Yaskawa INFORM job: TWIN_SKRZYNIA_5340_0_STOPNI_1OBR.JBI

/JOB
//NAME TWIN_SKRZYNIA_5340_0_STOPNI_1OBR
///FOLDERNAME 02-SKRZYNIE_JOBS
//POS
///NPOS 402,402,0,35,0,0
///TOOL 0
///POSTYPE PULSE
///PULSE
C00000=1055,-24125,84372,288,19725,204
C00001=1055,-24125,84372,288,19725,204
C00002=0,-15438,65714,0,-68532,0
C00003=25524,-25821,36823,19654,-58495,38520
C00004=23988,-24960,37134,18595,-57837,38812
C00005=22822,-23954,37534,17811,-57199,39017
C00006=22935,-24057,37491,17887,-57262,38997
C00007=20006,-24258,37408,15644,-56932,39751
C00008=24402,-25289,37013,18874,-58060,38740
C00009=22585,-24665,40358,17164,-59622,30036
C00010=23477,-23257,40205,18030,-58646,29630
C00011=22519,-22398,40568,17384,-58125,29795
C00012=22700,-22567,40495,17506,-58225,29764
C00013=19339,-22794,40398,14955,-57865,30607
C00014=24825,-24328,39798,18931,-59350,29401
C00015=32755,-32613,25711,29640,-48730,33694
C00016=25632,-30899,26166,23992,-46203,35378
C00017=24264,-29862,26497,22996,-45413,35639
C00018=24403,-29974,26459,23097,-45496,35612
C00019=20575,-30233,26374,19602,-44891,36810
C00020=26556,-31526,25988,24663,-46720,35206
C00021=30846,-32795,25752,28021,-48338,30427
C00022=24953,-30697,26306,23444,-45946,31743
C00023=23937,-29910,26558,22702,-45353,31936
C00024=24039,-29993,26530,22778,-45414,31916
C00025=20322,-30240,26449,19379,-44834,33080
C00026=25997,-31433,26093,24205,-46535,31545
C00027=26028,-43665,26580,-39946,8682,24640
C00028=27956,-30595,53065,-101898,6609,54413
C00029=26028,-43663,26580,-39944,8677,24639
C00030=38784,-34544,25404,33956,-51320,34445
C00031=29266,-32676,25756,26732,-47889,36488
C00032=25734,-31262,26119,24020,-46377,37252
C00033=24289,-30200,26441,22967,-45549,37525
C00034=24367,-30262,26420,23025,-45594,37511
C00035=20043,-30544,26331,19080,-44922,38860
C00036=26573,-31816,25967,24631,-46839,37095
C00037=27817,-32566,25782,25532,-47502,36865
C00038=25779,-31294,26110,24054,-46400,37243
C00039=24344,-30243,26427,23007,-45578,37515
C00040=24432,-30312,26405,23072,-45630,37498
C00041=20021,-30599,26315,19050,-44944,38872
C00042=26262,-31616,26021,24405,-46667,37153
C00043=27439,-32346,25835,25259,-47302,36935
C00044=25570,-31108,26163,23910,-46262,37277
C00045=24581,-30384,26384,23190,-45695,37464
C00046=24689,-30466,26358,23269,-45758,37444
C00047=20001,-30771,26264,18999,-45026,38899
C00048=26308,-31607,26026,24448,-46671,37139
C00049=27526,-32360,25834,25329,-47326,36914
C00050=24269,-40076,6479,29767,-34177,34232
C00051=22958,-37632,10123,27061,-35370,35326
C00052=22703,-41294,1722,31272,-29953,33282
C00053=19440,-41515,1663,27208,-29122,34832
C00054=25465,-43501,1200,33269,-31905,32752
C00055=87177,-39066,-1236,81808,-72661,19198
C00056=4794,-34097,38974,4189,-31824,-1302
C00057=4794,-34097,38974,4189,13412,-1302
C00058=11237,-37131,38982,-12694,5333,8253
C00059=6591,-33902,35532,5956,-1761,-1932
C00060=10065,-33530,28876,9373,-31104,-3154
C00061=31877,-32319,25770,29025,-48287,33360
C00062=24706,-30765,26196,23236,-45867,35119
C00063=23652,-29939,26460,22464,-45250,35320
C00064=23742,-30013,26436,22530,-45305,35302
C00065=19630,-30281,26348,18756,-44677,36597
C00066=26056,-31710,25928,24219,-46631,34863
C00067=38095,-40136,7813,41252,-44156,24924
C00068=33231,-38681,8176,37792,-41757,25918
C00069=31538,-37640,8473,36716,-40716,26179
C00070=31687,-37737,8444,36811,-40809,26155
C00071=27389,-38154,8322,32773,-39589,27627
C00072=33834,-39023,8084,38175,-42120,25821
C00073=4801,-35772,25187,4594,-28023,-1125
C00074=-1002,-39861,25115,1795,-37402,-69601
C00075=-1001,-39858,25114,1795,-37402,0
C00076=6591,-33902,35532,5956,-1761,-1932
C00077=6592,-33900,35531,103508,-35512,-26314
C00078=-99253,-13690,44082,59847,13407,-31313
C00079=-85045,-36869,-4353,28502,-22832,-52282
C00080=-92346,-18713,13565,21110,-22545,-55257
C00081=-85370,-14218,16934,32905,-23649,-60330
C00082=-84150,-13282,17685,34842,-23935,-61163
C00083=-82877,-12536,18624,36445,-24482,-61818
C00084=-83784,-13116,17825,35378,-24051,-61391
C00085=-85049,-11554,19196,33922,-23396,-60809
C00086=-84150,-13282,17685,34842,-23935,-61163
C00087=-85732,-21202,11427,30682,-24763,-59235
C00088=-84559,-15616,15722,33768,-24118,-60665
C00089=-84150,-13282,17685,34842,-23935,-61163
C00090=-83260,-12880,18034,36130,-24218,-61709
C00091=-84150,-13282,17685,34842,-23935,-61163
C00092=-85365,-11775,19006,33430,-23307,-60600
C00093=-84150,-13282,17685,34842,-23935,-61163
C00094=-85786,-16909,14677,31743,-23900,-59790
C00095=-84150,-13282,17685,34842,-23935,-61163
C00096=-83215,-12861,18051,36194,-24233,-61735
C00097=-84150,-13282,17685,34842,-23935,-61163
C00098=-85327,-11825,18959,33476,-23327,-60618
C00099=-84150,-13282,17685,34842,-23935,-61163
C00100=-87841,-18519,13420,28367,-23534,-58339
C00101=-84150,-13282,17685,34842,-23935,-61163
C00102=-83292,-12894,18020,36083,-24208,-61688
C00103=-84150,-13282,17685,34842,-23935,-61163
C00104=-85185,-12008,18799,33646,-23400,-60687
C00105=-84150,-13282,17685,34842,-23935,-61163
C00106=-86371,-18277,13606,30568,-23951,-59265
C00107=-84345,-13370,17612,34554,-23873,-61041
C00108=-83240,-12871,18042,36158,-24225,-61720
C00109=-84345,-13370,17612,34554,-23873,-61041
C00110=-85365,-12110,18711,33368,-23345,-60568
C00111=-84345,-13370,17612,34554,-23873,-61041
C00112=-86191,-19647,12567,30467,-24278,-59187
C00113=-84345,-13372,17610,34552,-23873,-61039
C00114=-83096,-12807,18098,36363,-24268,-61804
C00115=-84345,-13372,17610,34552,-23873,-61039
C00116=-85268,-12232,18600,33480,-23393,-60612
C00117=-84345,-13372,17610,34552,-23873,-61039
C00118=-84814,-16043,15376,33312,-24093,-60464
C00119=-84104,-13265,17702,34906,-23948,-61189
C00120=-82960,-12743,18153,36555,-24313,-61887
C00121=-84104,-13265,17702,34906,-23948,-61189
C00122=-84979,-12194,18635,33901,-23496,-60788
C00123=-84104,-13265,17702,34906,-23948,-61189
C00124=-86610,-16845,14732,30573,-23614,-59301
C00125=-84104,-13265,17702,34906,-23948,-61189
C00126=-82793,-12667,18222,36790,-24370,-61986
C00127=-84104,-13265,17702,34906,-23948,-61189
C00128=-84888,-12305,18537,34004,-23540,-60830
C00129=-84104,-13265,17702,34906,-23948,-61189
C00130=-83806,-19585,12613,33764,-25080,-60559
C00131=-83675,-13072,17868,35530,-24083,-61453
C00132=-82553,-12556,18319,37130,-24451,-62127
C00133=-83675,-13072,17868,35530,-24083,-61453
C00134=-84378,-12223,18610,34735,-23716,-61138
C00135=-83675,-13072,17868,35530,-24083,-61453
C00136=-87149,-17993,13826,29513,-23647,-58830
C00137=-84104,-13265,17702,34906,-23948,-61189
C00138=-82640,-12594,18285,37014,-24425,-62079
C00139=-84104,-13265,17702,34906,-23948,-61189
C00140=-84792,-12429,18430,34119,-23592,-60877
C00141=-84104,-13265,17702,34906,-23948,-61189
C00142=-83583,-9185,30892,23668,-36042,-57025
C00143=-85789,-8328,35795,20592,-37093,-55378
C00144=-85786,-16735,14816,31782,-23869,-59812
C00145=-84103,-13263,17702,34906,-23947,-61191
C00146=-83225,-12865,18046,36177,-24227,-61729
C00147=-84103,-13263,17702,34906,-23947,-61191
C00148=-84774,-12447,18412,34138,-23599,-60886
C00149=-84103,-13263,17702,34906,-23947,-61191
C00150=-86149,-16246,6730,18897,-35239,-57128
C00151=-86244,-15289,7532,18875,-35060,-57127
C00152=-85361,-14893,7870,19824,-35193,-57574
C00153=-86244,-15289,7532,18875,-35060,-57127
C00154=-86889,-14409,8282,18264,-34784,-56850
C00155=-86244,-15289,7532,18875,-35060,-57127
C00156=-90262,-21765,2389,14114,-35574,-54847
C00157=-90262,-21765,2389,28730,-17672,-54847
C00158=-89967,-19086,25635,28730,-17672,-54847
C00159=568,-24029,84339,168,19981,112
C00160=568,-24677,83015,164,20405,113
C00161=101153,-24598,83176,165,20353,113
C00162=101153,-24598,83176,165,20353,113
C00163=89967,-19086,25635,-28730,-17672,54847
C00164=90262,-21765,2389,-28730,-17672,54847
C00165=86932,-18662,4771,-17876,-35519,56628
C00166=86578,-15436,7408,-18515,-35011,56957
C00167=85428,-14922,7844,-19753,-35183,57541
C00168=84405,-14447,8250,-20842,-35348,58054
C00169=85428,-14922,7844,-19753,-35183,57541
C00170=86134,-13973,8661,-19091,-34881,57237
C00171=85428,-14922,7844,-19753,-35183,57541
C00172=85786,-16735,14816,-31782,-23869,59812
C00173=83514,-12996,17929,-35760,-24132,61552
C00174=82296,-12429,18424,-37488,-24534,62281
C00175=83514,-12996,17929,-35760,-24132,61552
C00176=84266,-12085,18725,-34910,-23738,61214
C00177=83514,-12996,17929,-35760,-24132,61552
C00178=87323,-6914,39851,-18853,-38149,44508
C00179=83118,-12818,18089,-36330,-24263,61791
C00180=81969,-12276,18566,-37944,-24648,62472
C00181=83118,-12818,18089,-36330,-24263,61791
C00182=83927,-11846,18941,-35423,-23842,61433
C00183=83118,-12818,18089,-36330,-24263,61791
C00184=83806,-19585,12613,-33764,-25080,60559
C00185=83148,-12832,18077,-36287,-24254,61773
C00186=81889,-12236,18598,-38058,-24676,62520
C00187=83148,-12832,18077,-36287,-24254,61773
C00188=83900,-11930,18867,-35446,-23862,61440
C00189=83148,-12832,18077,-36287,-24254,61773
C00190=86610,-16845,14732,-30573,-23614,59301
C00191=82493,-13239,17725,-37070,-24559,62089
C00192=81442,-12739,18159,-38529,-24915,62703
C00193=82493,-13239,17725,-37070,-24559,62089
C00194=83435,-12133,18689,-36040,-24063,61682
C00195=82493,-13239,17725,-37070,-24559,62089
C00196=84814,-16043,15376,-33312,-24093,60464
C00197=82555,-13613,17404,-36910,-24580,62015
C00198=81369,-13053,17885,-38558,-24979,62709
C00199=82555,-13613,17404,-36910,-24580,62015
C00200=83568,-12431,18429,-35805,-24046,61580
C00201=82555,-13613,17404,-36910,-24580,62015
C00202=86191,-19647,12567,-30467,-24278,59187
C00203=82500,-13648,17375,-36975,-24607,62039
C00204=81594,-13224,17740,-38236,-24911,62571
C00205=82500,-13648,17375,-36975,-24607,62039
C00206=83449,-12543,18332,-35941,-24104,61633
C00207=82500,-13648,17375,-36975,-24607,62039
C00208=86371,-18277,13606,-30568,-23951,59265
C00209=82904,-13790,17251,-36416,-24470,61808
C00210=81796,-13275,17692,-37971,-24838,62464
C00211=82904,-13790,17251,-36416,-24470,61808
C00212=83696,-12867,18046,-35547,-24051,61466
C00213=82904,-13790,17251,-36416,-24470,61808
C00214=87841,-18519,13420,-28367,-23534,58339
C00215=82748,-13879,17174,-36603,-24542,61883
C00216=81789,-13434,17554,-37946,-24861,62449
C00217=82748,-13879,17174,-36603,-24542,61883
C00218=83603,-12888,18026,-35668,-24086,61514
C00219=82748,-13879,17174,-36603,-24542,61883
C00220=85786,-16909,14677,-31743,-23900,59790
C00221=82339,-14116,16972,-37087,-24733,62079
C00222=81557,-13752,17280,-38171,-24994,62536
C00223=82339,-14116,16972,-37087,-24733,62079
C00224=83390,-12909,18006,-35951,-24172,61633
C00225=82339,-14116,16972,-37087,-24733,62079
C00226=85732,-21202,11427,-30682,-24763,59235
C00227=82398,-14365,16763,-36952,-24745,62014
C00228=81340,-13876,17176,-38416,-25096,62632
C00229=82398,-14365,16763,-36952,-24745,62014
C00230=83629,-12951,17972,-35620,-24090,61491
C00231=82398,-14365,16763,-36952,-24745,62014
C00232=92346,-18713,13565,-21110,-22545,55257
C00233=82794,-13980,17083,-36511,-24538,61844
C00234=81697,-13472,17516,-38043,-24902,62488
C00235=82794,-13980,17083,-36511,-24538,61844
C00236=83767,-12847,18056,-35444,-24023,61424
C00237=82794,-13980,17083,-36511,-24538,61844
C00238=85045,-36869,-4353,-28502,-22832,52282
C00239=69856,-53931,-13446,-33557,-28911,29591
C00240=73943,-28815,39553,-16801,-45089,19004
C00241=73943,-28815,39553,-16801,-45089,19004
C00242=0,-24029,84339,0,19981,0
C00243=0,-24029,84339,0,19981,0
C00244=0,-52280,40443,0,6876,0
C00245=63961,-36661,14391,66570,-58199,13439
C00246=50233,-31965,16595,55443,-54435,15843
C00247=47147,-32819,12541,55607,-51124,17230
C00248=46896,-37872,871,62973,-46008,11193
C00249=54160,-39955,137,66075,-50361,10746
C00250=0,-52280,40443,0,6876,0
C00251=0,-52280,40443,1,6876,0
C00252=42978,-45587,7631,48214,-41849,18034
C00253=34615,-32719,24207,35617,-45539,22507
C00254=46734,-24688,30880,50025,-55713,21863
C00255=45059,-39151,-3508,69830,-41334,11649
C00256=32474,-45233,-13338,65386,-28486,22104
C00257=59828,-44646,-5405,72855,-48572,12139
C00258=0,-38761,66314,0,-763,0
C00259=0,-44757,54667,0,2744,0
C00260=40382,-38226,12225,48505,-40693,16039
C00261=55481,-27484,23768,62968,-54833,11978
C00262=49796,-26552,24209,59898,-51910,12564
C00263=49435,-31346,12259,54968,-55893,13137
C00264=55330,-33748,11238,57660,-59334,12681
C00265=78664,-24436,10378,82837,-79111,12029
C00266=75189,-23065,11287,81851,-76948,11927
C00267=75189,-45249,11287,81851,-38847,11927
C00268=29880,-45249,11287,43145,-11324,11927
C00269=0,-24029,84339,0,19981,0
C00270=0,-24026,84338,1,19977,2
C00271=4264,-34194,25387,4006,-26954,-29436
C00272=1,-24024,84337,2,19973,1
C00273=1,-24024,84337,2,19973,1
C00274=3796,-57671,22373,2336,-25309,-753
C00275=52632,-34554,16626,51161,-63050,5622
C00276=59461,-32779,9832,66317,-58406,17312
C00277=52698,-27865,19111,60288,-56542,14852
C00278=51544,-17445,41630,51689,-64712,19351
C00279=62932,-33588,12189,66848,-61063,18031
C00280=1,-24024,84337,2,19973,1
C00281=1,-24024,84337,2,19973,1
C00282=57188,-41777,19973,48132,-58706,4905
C00283=55566,-48748,-16991,79805,-45048,-6941
C00284=49908,-48716,-25784,90749,-41340,-3650
C00285=44252,-47412,-25530,90709,-37744,-4391
C00286=43421,-46995,-25379,90839,-37219,-4572
C00287=55479,-50244,-26473,91085,-44870,-3042
C00288=12119,-24859,71505,13236,4440,2633
C00289=-91085,-34291,10385,1908,-24348,-42097
C00290=-86191,-19647,12567,30467,-24278,-59187
C00291=-99148,-11667,19101,-13975,-20192,-40187
C00292=-98206,-11518,19604,-10142,-20308,-41629
C00293=-99474,-20389,12397,-11593,-22150,-41069
C00294=0,-52280,40443,0,6876,0
C00295=85348,-24204,23536,-13963,-15515,44275
C00296=84670,-17015,14597,-33277,-24304,60423
C00297=96971,-12584,18294,8365,-19955,42614
C00298=97182,-12918,18001,8747,-20027,42449
C00299=96230,-24528,9149,6144,-22576,43630
C00300=0,-52280,40443,0,6876,0
C00301=0,-52280,40443,0,6876,0
C00302=-90140,-60305,18108,-2708,1721,-7625
C00303=-95594,-27428,6866,-4663,-19832,-42154
C00304=-99356,-13410,18355,-15385,-17730,-37479
C00305=-99405,-10878,20508,-15853,-17333,-37255
C00306=-99132,-10804,20575,-15274,-17279,-37502
C00307=-99132,-3482,39129,-10940,-24351,-39674
C00308=-98851,-3328,38974,-10588,-24101,-39807
C00309=-100183,-18601,14070,-16273,-18800,-37146
C00310=-90140,-60305,18108,-2708,1721,-7625
C00311=0,-52280,40443,0,6876,0
C00312=84259,-57935,27522,-3761,3673,6310
C00313=86507,-39672,4297,-27618,-16640,46340
C00314=70477,-27878,7073,-45786,-32339,64941
C00315=84043,-16293,15174,-34312,-24409,60872
C00316=94507,-13191,17794,-563,-19874,46473
C00317=99154,-17369,4403,32227,-9753,28926
C00318=99154,-17369,4403,32227,-9753,28926
C00319=98946,-17182,4556,31649,-9649,29182
C00320=100388,-17987,13832,15751,-21517,39479
C00321=86507,-39672,4297,-27618,-16640,46340
C00322=84259,-57935,27522,-3761,3673,6310
C00323=0,-52280,40443,0,6876,0
C00324=0,-27933,77061,0,20812,0
C00325=0,-27933,77061,0,20812,0
C00326=0,-52280,40443,0,6876,0
C00327=-91970,-60791,14435,-3343,512,-9412
C00328=-99196,-15868,16098,-13748,-19297,-38710
C00329=-99196,-15868,16098,-13748,-19297,-38710
C00330=-99196,-15868,16098,-13748,-19297,-38710
C00331=-85815,-11758,19597,31748,-21097,-58265
C00332=-87383,-11883,19487,26986,-20206,-56250
C00333=-99562,-16264,15781,-14410,-19427,-38431
C00334=-99196,-15868,16098,-13748,-19297,-38710
C00335=-91970,-60791,14435,-3343,512,-9412
C00336=0,-52280,40443,0,6876,0
C00337=91083,-60784,14823,-9043,-825,15173
C00338=83869,-19403,12921,-33769,-24740,60260
C00339=83869,-19403,12921,-33769,-24740,60260
C00340=83420,-14897,16486,-35538,-24144,61113
C00341=90535,-11845,19652,-14037,-20800,51549
C00342=90317,-11662,19878,-14346,-20882,51648
C00343=95871,-14889,15992,4901,-19605,43825
C00344=83869,-19403,12921,-33769,-24740,60260
C00345=91083,-60784,14823,-9043,-825,15173
C00346=0,-52280,40443,0,6876,0
C00347=-91526,-60598,16699,7584,176,-13289
C00348=-94392,-6553,48683,5805,-47321,-49764
C00349=-88951,-345,54953,10686,-47392,-51569
C00350=-88172,5833,62122,11322,-47753,-51785
C00351=-90949,-14015,9500,8834,-34399,-51934
C00352=-84917,-15593,15742,33275,-23984,-60461
C00353=-81669,-15982,15425,37506,-25258,-62202
C00354=-79867,-25377,9541,37586,-25936,-59971
C00355=-91415,-60262,16631,7870,-73,-13734
C00356=24,-24029,84339,7,19981,5
C00357=160,-24029,84339,47,19981,32
C00358=99096,-24029,84339,47,19981,32
C00359=99096,-24029,84339,47,19981,32
C00360=89967,-19086,25635,-28730,-17672,54847
C00361=85786,-16735,14816,-31782,-23869,59812
C00362=83492,-14473,16674,-35480,-24338,61406
C00363=82709,-11470,19305,-37370,-24374,62232
C00364=85293,-13629,8874,-19696,-34851,57583
C00365=85505,-16299,6686,-19564,-35388,57437
C00366=89967,-19086,25635,-28730,-17672,54847
C00367=568,-24029,84339,168,19981,112
C00368=568,-24029,84339,168,19981,112
C00369=-91970,-60791,14435,-3343,512,-9412
C00370=-86948,-23217,10819,28314,-23349,-56438
C00371=-85895,-16522,15767,31843,-22281,-58087
C00372=-93643,1708,52973,2937,-38210,-34777
C00373=-93409,-737,47229,3345,-36106,-34967
C00374=-86145,-24679,9854,29028,-23971,-56682
C00375=-100471,-58311,4157,14142,-4822,-27614
C00376=-68517,-58311,4157,14142,-4822,-27614
C00377=0,-52280,40443,0,6876,0
C00378=91083,-60784,14823,-9043,-825,15173
C00379=83869,-19403,12921,-33769,-24740,60260
C00380=82620,-18743,14708,-32942,-26226,58979
C00381=83315,-11405,20766,-33572,-24860,59408
C00382=83326,-11144,20997,-33599,-24827,59423
C00383=84798,-22668,11879,-29033,-26372,57255
C00384=91083,-60784,14823,-9043,-825,15173
C00385=0,-52280,40443,0,6876,0
C00386=-6369,-39206,65423,-4801,-482,2563
C00387=-97287,-29142,12714,-8673,-22288,-37832
C00388=-86191,-19647,12567,30467,-24278,-59187
C00389=-85671,-16302,15857,30808,-24404,-58999
C00390=-99965,-10410,22406,-14600,-22538,-38834
C00391=-95758,-10871,21797,-1120,-21702,-44724
C00392=-87910,-17792,15835,25414,-24996,-56048
C00393=-97287,-29142,12714,-8673,-22288,-37832
C00394=0,-52280,40443,0,6876,0
C00395=92301,-25634,22749,2368,-15645,37646
C00396=83738,-18329,13570,-34202,-24868,60772
C00397=90096,-13099,18146,-15422,-20883,52700
C00398=93330,-13245,17928,-4627,-20146,48105
C00399=80226,-20465,12178,-39626,-27411,62762
C00400=92301,-25634,22749,2368,-15645,37646
C00401=0,-52280,40443,0,6876,0
BC00000=413138
BC00001=413138
BC00002=413138
BC00003=413134
BC00004=413134
BC00005=413134
BC00006=413134
BC00007=413134
BC00008=413134
BC00009=474623
BC00010=474628
BC00011=474628
BC00012=474628
BC00013=474628
BC00014=474628
BC00015=522849
BC00016=522849
BC00017=522849
BC00018=522849
BC00019=522849
BC00020=522849
BC00021=586045
BC00022=586045
BC00023=586045
BC00024=586045
BC00025=586045
BC00026=586045
BC00027=479622
BC00028=618860
BC00029=673957
BC00030=663090
BC00031=663090
BC00032=663090
BC00033=663090
BC00034=663090
BC00035=663090
BC00036=663090
BC00037=708270
BC00038=708270
BC00039=708270
BC00040=708270
BC00041=708270
BC00042=708270
BC00043=770184
BC00044=770184
BC00045=770184
BC00046=770184
BC00047=770184
BC00048=770184
BC00049=823730
BC00050=829967
BC00051=829969
BC00052=829970
BC00053=829970
BC00054=829970
BC00055=838761
BC00056=740349
BC00057=687700
BC00058=771943
BC00059=861898
BC00060=900223
BC00061=904141
BC00062=901229
BC00063=901229
BC00064=901229
BC00065=901229
BC00066=901229
BC00067=949836
BC00068=949836
BC00069=949836
BC00070=949836
BC00071=949836
BC00072=965197
BC00073=941874
BC00074=915598
BC00075=930961
BC00076=861898
BC00077=861901
BC00078=861901
BC00079=931504
BC00080=963634
BC00081=963631
BC00082=963631
BC00083=963631
BC00084=963631
BC00085=963631
BC00086=963631
BC00087=902188
BC00088=902188
BC00089=902188
BC00090=902188
BC00091=902188
BC00092=902188
BC00093=902188
BC00094=840744
BC00095=840744
BC00096=840744
BC00097=840744
BC00098=840744
BC00099=840744
BC00100=779300
BC00101=779300
BC00102=779300
BC00103=779300
BC00104=779300
BC00105=779300
BC00106=717855
BC00107=717855
BC00108=717855
BC00109=717855
BC00110=717855
BC00111=717855
BC00112=656405
BC00113=656405
BC00114=656405
BC00115=656405
BC00116=656405
BC00117=656405
BC00118=594961
BC00119=594961
BC00120=594961
BC00121=594961
BC00122=594961
BC00123=594961
BC00124=533517
BC00125=533517
BC00126=533517
BC00127=533517
BC00128=533517
BC00129=533517
BC00130=472073
BC00131=472073
BC00132=472073
BC00133=472073
BC00134=472073
BC00135=472073
BC00136=410629
BC00137=410629
BC00138=410629
BC00139=410629
BC00140=410629
BC00141=410629
BC00142=410629
BC00143=349186
BC00144=349186
BC00145=349186
BC00146=349186
BC00147=349186
BC00148=349186
BC00149=349186
BC00150=336469
BC00151=336469
BC00152=336469
BC00153=336469
BC00154=336469
BC00155=336469
BC00156=336469
BC00157=336469
BC00158=336469
BC00159=336469
BC00160=511557
BC00161=512005
BC00162=363797
BC00163=336469
BC00164=336469
BC00165=337415
BC00166=337415
BC00167=337415
BC00168=337415
BC00169=337415
BC00170=337415
BC00171=337415
BC00172=349186
BC00173=350137
BC00174=350137
BC00175=350137
BC00176=350137
BC00177=350137
BC00178=410629
BC00179=411580
BC00180=411580
BC00181=411580
BC00182=411580
BC00183=411580
BC00184=472073
BC00185=473025
BC00186=473025
BC00187=473025
BC00188=473025
BC00189=473025
BC00190=533517
BC00191=534468
BC00192=534468
BC00193=534468
BC00194=534468
BC00195=534468
BC00196=594961
BC00197=594961
BC00198=594961
BC00199=594961
BC00200=594961
BC00201=594961
BC00202=656405
BC00203=657350
BC00204=657350
BC00205=657350
BC00206=657350
BC00207=657350
BC00208=717855
BC00209=718799
BC00210=718799
BC00211=718799
BC00212=718799
BC00213=718799
BC00214=779300
BC00215=780245
BC00216=780245
BC00217=780245
BC00218=780245
BC00219=780245
BC00220=840744
BC00221=841691
BC00222=841691
BC00223=841691
BC00224=841691
BC00225=841691
BC00226=902188
BC00227=903136
BC00228=903136
BC00229=903136
BC00230=903136
BC00231=903136
BC00232=963634
BC00233=963633
BC00234=963633
BC00235=963633
BC00236=963633
BC00237=963633
BC00238=931504
BC00239=861901
BC00240=861901
BC00241=881624
BC00242=769966
BC00243=769966
BC00244=716865
BC00245=668657
BC00246=668657
BC00247=668657
BC00248=717171
BC00249=717171
BC00250=716865
BC00251=800897
BC00252=908887
BC00253=899019
BC00254=895607
BC00255=945882
BC00256=955598
BC00257=945882
BC00258=840120
BC00259=538973
BC00260=485226
BC00261=456696
BC00262=456696
BC00263=417276
BC00264=417276
BC00265=493986
BC00266=514306
BC00267=514306
BC00268=514306
BC00269=493986
BC00270=797003
BC00271=895791
BC00272=812362
BC00273=476651
BC00274=522561
BC00275=566531
BC00276=593948
BC00277=593948
BC00278=529848
BC00279=529848
BC00280=461290
BC00281=663315
BC00282=778314
BC00283=778312
BC00284=778312
BC00285=778312
BC00286=838222
BC00287=838222
BC00288=566410
BC00289=679663
BC00290=656405
BC00291=656405
BC00292=717855
BC00293=717855
BC00294=717855
BC00295=662303
BC00296=657350
BC00297=657350
BC00298=718803
BC00299=718803
BC00300=717855
BC00301=792672
BC00302=792672
BC00303=896850
BC00304=895720
BC00305=895720
BC00306=957178
BC00307=957178
BC00308=978461
BC00309=957178
BC00310=792672
BC00311=792672
BC00312=792672
BC00313=887446
BC00314=903126
BC00315=903126
BC00316=903126
BC00317=964577
BC00318=976097
BC00319=993812
BC00320=964577
BC00321=887446
BC00322=792672
BC00323=792672
BC00324=700249
BC00325=546214
BC00326=546214
BC00327=546211
BC00328=546211
BC00329=406776
BC00330=406776
BC00331=406778
BC00332=468200
BC00333=468200
BC00334=546211
BC00335=546211
BC00336=546214
BC00337=546214
BC00338=507604
BC00339=410782
BC00340=410782
BC00341=410782
BC00342=472720
BC00343=472720
BC00344=507604
BC00345=546214
BC00346=546214
BC00347=516757
BC00348=383716
BC00349=349186
BC00350=349186
BC00351=336469
BC00352=349186
BC00353=410629
BC00354=416512
BC00355=515801
BC00356=520018
BC00357=474013
BC00358=474013
BC00359=403108
BC00360=336469
BC00361=349186
BC00362=349186
BC00363=349186
BC00364=337415
BC00365=337415
BC00366=336469
BC00367=336469
BC00368=428401
BC00369=546211
BC00370=591088
BC00371=591088
BC00372=591088
BC00373=531116
BC00374=529640
BC00375=529640
BC00376=529640
BC00377=529640
BC00378=546214
BC00379=589919
BC00380=595627
BC00381=595627
BC00382=534177
BC00383=534177
BC00384=546214
BC00385=529640
BC00386=651195
BC00387=765890
BC00388=777968
BC00389=778453
BC00390=779252
BC00391=840748
BC00392=840748
BC00393=765890
BC00394=717855
BC00395=741100
BC00396=780224
BC00397=780222
BC00398=841743
BC00399=841743
BC00400=741100
BC00401=717855
///POSTYPE BASE
///RECTAN
///RCONF 0,0,0,0,0,0,0,0,0,0,0,0,0,0,0,0,0,0,0,0,0,0,0,0
P00006=-2.449,0.031,8.825,0.0000,0.0000,0.0000
///RCONF 1,0,0,0,0,0,0,0,0,0,0,0,0,0,0,0,0,0,0,0,0,0,0,0
P00100=-0.081,2.558,4.482,0.0000,0.0000,0.0000
P00101=0.030,-2.286,2.993,0.0000,0.0000,0.0000
P00102=-0.005,-1.108,1.644,0.0000,0.0000,0.0000
P00103=-0.094,-3.400,4.200,0.0000,0.0000,0.0000
P00104=0.043,-2.127,5.826,0.0000,0.0000,0.0000
P00105=-0.043,0.662,5.286,0.0000,0.0000,0.0000
P00106=-0.018,-2.519,0.237,0.0000,0.0000,0.0000
P00107=-0.008,-4.537,-4.500,0.0000,0.0000,0.0000
P00108=0.014,-3.040,2.637,0.0000,0.0000,0.0000
P00109=0.017,-3.622,2.341,0.0000,0.0000,0.0000
P00300=-0.036,-1.505,2.318,0.0000,0.0000,0.0000
///RCONF 0,0,0,0,0,0,0,0,0,0,0,0,0,0,0,0,0,0,0,0,0,0,0,0
P00301=0.005,-4.708,-4.628,0.0000,0.0000,0.0000
P00302=0.052,-2.937,-4.426,0.0000,0.0000,0.0000
P00303=-0.004,-1.437,-4.584,0.0000,0.0000,0.0000
P00304=0.028,-1.666,-4.234,0.0000,0.0000,0.0000
P00305=-0.003,-1.920,-3.501,0.0000,0.0000,0.0000
P00306=0.015,-2.252,-3.054,0.0000,0.0000,0.0000
P00307=0.019,-2.151,-5.077,0.0000,0.0000,0.0000
P00308=-0.003,-2.092,-4.888,0.0000,0.0000,0.0000
P00309=-0.040,-2.205,-4.992,0.0000,0.0000,0.0000
P00310=-0.006,-2.490,-5.925,0.0000,0.0000,0.0000
P00311=-0.007,-2.079,-5.307,0.0000,0.0000,0.0000
P00350=11.519,-0.008,1.149,0.0000,0.0000,0.0000
P00351=13.563,-0.027,-0.653,0.0000,0.0000,0.0000
P00352=13.252,-0.027,-0.827,0.0000,0.0000,0.0000
P00353=10.971,-0.082,0.776,0.0000,0.0000,0.0000
P00354=-0.024,2.508,-1.824,0.0000,0.0000,0.0000
P00355=-0.001,2.528,-1.131,0.0000,0.0000,0.0000
P00356=-0.034,2.921,-0.262,0.0000,0.0000,0.0000
P00357=0.003,3.386,-0.091,0.0000,0.0000,0.0000
P00358=0.014,3.037,-0.020,0.0000,0.0000,0.0000
P00359=-0.005,2.731,0.912,0.0000,0.0000,0.0000
P00360=-0.011,3.412,0.438,0.0000,0.0000,0.0000
P00361=0.018,3.050,1.253,0.0000,0.0000,0.0000
//INST
///DATE 2024/12/12 11:36
///ATTR SC,RW
///GROUP1 RB1,BS1
NOP
CALL JOB:MOVE_INTO_TUNNEL
MOVJ C00000 BC00000 VJ=30.00
'------------------------
'------------------------
'SPOINA SRODEK DOL
'------------------------
'------------------------
'POMIAR DO WYJ!! PRZEROBIC NA STD
MOVJ C00001 BC00001 VJ=40.00
MOVJ C00002 BC00002 VJ=40.00
'W3P
MOVJ C00003 BC00003 VJ=20.00 PL=0
MOVL C00004 BC00004 V=166.7 PL=0
REFP 3 C00005 BC00005
CALL JOB:SEARCH-R1
SET P0100 P0006
SFTON P0100
MOVL C00006 BC00006 V=66.7 PL=0
REFP 3 C00007 BC00007
CALL JOB:SEARCH-R1
SET P0100 P0006
SFTON P0100
MOVL C00008 BC00008 V=333.3 PL=0
SFTOF
'W3L
MOVL C00009 BC00009 V=666.7
MOVL C00010 BC00010 V=166.7 PL=0
REFP 3 C00011 BC00011
CALL JOB:SEARCH-R1
SET P0101 P0006
SFTON P0101
MOVL C00012 BC00012 V=166.7 PL=0
REFP 3 C00013 BC00013
CALL JOB:SEARCH-R1
SET P0101 P0006
SFTON P0101
MOVL C00014 BC00014 V=333.3 PL=0
SFTOF
'W9P
MOVL C00015 BC00015 V=666.7
MOVL C00016 BC00016 V=166.7
REFP 3 C00017 BC00017
CALL JOB:SEARCH-R1
SET P0102 P0006
SFTON P0102
MOVL C00018 BC00018 V=166.7 PL=0
REFP 3 C00019 BC00019
CALL JOB:SEARCH-R1
SET P0102 P0006
SFTON P0102
MOVL C00020 BC00020 V=333.3 PL=0
'W9L
MOVL C00021 BC00021 V=666.7
MOVL C00022 BC00022 V=166.7
REFP 3 C00023 BC00023
CALL JOB:SEARCH-R1
SET P0103 P0006
SFTON P0103
MOVL C00024 BC00024 V=166.7 PL=0
REFP 3 C00025 BC00025
CALL JOB:SEARCH-R1
SET P0103 P0006
SFTON P0103
MOVL C00026 BC00026 V=333.3 PL=0
'PRZEJAZ NAD BELKA
MOVL C00027 BC00027 V=666.7
MOVJ C00028 BC00028 VJ=40.00
MOVJ C00029 BC00029 VJ=40.00
MOVJ C00030 BC00030 VJ=40.00
'W1P
MOVJ C00031 BC00031 VJ=20.00 PL=0
MOVL C00032 BC00032 V=166.7 PL=0
REFP 3 C00033 BC00033
CALL JOB:SEARCH-R1
SET P0104 P0006
SFTON P0104
MOVL C00034 BC00034 V=166.7 PL=0
REFP 3 C00035 BC00035
CALL JOB:SEARCH-R1
SET P0104 P0006
SFTON P0104
MOVL C00036 BC00036 V=333.3 PL=0
SFTOF
'W1L
MOVL C00037 BC00037 V=666.7
MOVL C00038 BC00038 V=166.7 PL=0
REFP 3 C00039 BC00039
CALL JOB:SEARCH-R1
SET P0105 P0006
SFTON P0105
MOVL C00040 BC00040 V=166.7 PL=0
REFP 3 C00041 BC00041
CALL JOB:SEARCH-R1
SET P0105 P0006
SFTON P0105
MOVL C00042 BC00042 V=333.3 PL=0
SFTOF
MOVL C00043 BC00043 V=666.7
'W10P
MOVL C00044 BC00044 V=166.7 PL=0
REFP 3 C00045 BC00045
CALL JOB:SEARCH-R1
SET P0106 P0006
SFTON P0106
MOVL C00046 BC00046 V=166.7 PL=0
REFP 3 C00047 BC00047
CALL JOB:SEARCH-R1
SET P0106 P0006
SFTON P0106
MOVL C00048 BC00048 V=333.3 PL=0
SFTOF
'W10L
MOVL C00049 BC00049 V=333.3
MOVL C00050 BC00050 V=166.7 PL=0
REFP 3 C00051 BC00051
CALL JOB:SEARCH-R1
SET P0107 P0006
SFTON P0107
MOVL C00052 BC00052 V=166.7 PL=0
REFP 3 C00053 BC00053
CALL JOB:SEARCH-R1
SET P0107 P0006
SFTON P0107
MOVL C00054 BC00054 V=333.3 PL=0
SFTOF
MOVL C00055 BC00055 V=333.3
'PRZEJAZD
MOVJ C00056 BC00056 VJ=50.00
MOVJ C00057 BC00057 VJ=50.00
MOVJ C00058 BC00058 VJ=60.00
MOVJ C00059 BC00059 VJ=60.00
MOVJ C00060 BC00060 VJ=60.00
MOVJ C00061 BC00061 VJ=60.00 PL=0
MOVL C00062 BC00062 V=166.7 PL=0
REFP 3 C00063 BC00063
CALL JOB:SEARCH-R1
SET P0108 P0006
SFTON P0108
MOVL C00064 BC00064 V=166.7 PL=0
REFP 3 C00065 BC00065
CALL JOB:SEARCH-R1
SET P0108 P0006
SFTON P0108
MOVL C00066 BC00066 V=333.3 PL=0
SFTOF
'W2P
'W2L
MOVL C00067 BC00067 V=666.7
MOVL C00068 BC00068 V=166.7 PL=0
REFP 3 C00069 BC00069
CALL JOB:SEARCH-R1
SET P0109 P0006
SFTON P0109
MOVL C00070 BC00070 V=166.7 PL=0
REFP 3 C00071 BC00071
CALL JOB:SEARCH-R1
SET P0109 P0006
SFTON P0109
MOVL C00072 BC00072 V=333.3 PL=0
MOVJ C00073 BC00073 VJ=20.00
SFTOF
CALL JOB:TWIN_5340_0ST_RAMA_PRZ_OBR1_POM
'.................
'.................
'.................
'PROG POMIARY RAMA PRZED
'.................
'.................
'.................
MOVJ C00074 BC00074 VJ=50.00
'------------------------
'------------------------
'PRAWA STRONA PROFIL GORA
'------------------------
'------------------------
MOVJ C00075 BC00075 VJ=50.00
MOVJ C00076 BC00076 VJ=50.00
MOVJ C00077 BC00077 VJ=50.00
MOVJ C00078 BC00078 VJ=20.00
MOVJ C00079 BC00079 VJ=50.00
'------------------------
'W14A L
'------------------------
SFTOF
MOVJ C00080 BC00080 VJ=50.00
MOVJ C00081 BC00081 VJ=30.00
MOVL C00082 BC00082 V=166.7 PL=0
REFP 3 C00083 BC00083
CALL JOB:SEARCH-R1
SET P0300 P0006
SFTON P0300
MOVL C00084 BC00084 V=166.7 PL=0
REFP 3 C00085 BC00085
CALL JOB:SEARCH-R1
SET P0300 P0006
SFTON P0300
MOVL C00086 BC00086 V=166.7 PL=0
SFTOF
'------------------------
'W14A P
'------------------------
SFTOF
MOVJ C00087 BC00087 VJ=50.00
MOVJ C00088 BC00088 VJ=50.00
MOVL C00089 BC00089 V=166.7 PL=0
REFP 3 C00090 BC00090
CALL JOB:SEARCH-R1
SET P0301 P0006
SFTON P0301
MOVL C00091 BC00091 V=166.7 PL=0
REFP 3 C00092 BC00092
CALL JOB:SEARCH-R1
SET P0301 P0006
SFTON P0301
MOVL C00093 BC00093 V=166.7 PL=0
SFTOF
'------------------------
'W19A L
'------------------------
SFTOF
MOVJ C00094 BC00094 VJ=50.00
MOVL C00095 BC00095 V=200.0 PL=0
REFP 3 C00096 BC00096
CALL JOB:SEARCH-R1
SET P0302 P0006
SFTON P0302
MOVL C00097 BC00097 V=166.7 PL=0
REFP 3 C00098 BC00098
CALL JOB:SEARCH-R1
SET P0302 P0006
SFTON P0302
MOVL C00099 BC00099 V=250.0 PL=0
SFTOF
'------------------------
'W19A P
'------------------------
SFTOF
MOVJ C00100 BC00100 VJ=50.00
MOVL C00101 BC00101 V=166.7 PL=0
REFP 3 C00102 BC00102
CALL JOB:SEARCH-R1
SET P0303 P0006
SFTON P0303
MOVL C00103 BC00103 V=166.7 PL=0
REFP 3 C00104 BC00104
CALL JOB:SEARCH-R1
SET P0303 P0006
SFTON P0303
MOVL C00105 BC00105 V=166.7 PL=0
SFTOF
'------------------------
'W13A L
'------------------------
SFTOF
MOVJ C00106 BC00106 VJ=50.00
MOVL C00107 BC00107 V=166.7 PL=0
REFP 3 C00108 BC00108
CALL JOB:SEARCH-R1
SET P0304 P0006
SFTON P0304
MOVL C00109 BC00109 V=166.7 PL=0
REFP 3 C00110 BC00110
CALL JOB:SEARCH-R1
SET P0304 P0006
SFTON P0304
MOVL C00111 BC00111 V=166.7 PL=0
SFTOF
'------------------------
'W13A P
'------------------------
SFTOF
MOVJ C00112 BC00112 VJ=50.00
MOVL C00113 BC00113 V=200.0 PL=0
REFP 3 C00114 BC00114
CALL JOB:SEARCH-R1
SET P0305 P0006
SFTON P0305
MOVL C00115 BC00115 V=166.7 PL=0
REFP 3 C00116 BC00116
CALL JOB:SEARCH-R1
SET P0305 P0006
SFTON P0305
MOVL C00117 BC00117 V=250.0 PL=0
SFTOF
'------------------------
'W18A L
'------------------------
SFTOF
MOVJ C00118 BC00118 VJ=50.00
MOVL C00119 BC00119 V=200.0 PL=0
REFP 3 C00120 BC00120
CALL JOB:SEARCH-R1
SET P0306 P0006
SFTON P0306
MOVL C00121 BC00121 V=166.7 PL=0
REFP 3 C00122 BC00122
CALL JOB:SEARCH-R1
SET P0306 P0006
SFTON P0306
MOVL C00123 BC00123 V=166.7 PL=0
SFTOF
'------------------------
'W18A P
'------------------------
SFTOF
MOVJ C00124 BC00124 VJ=50.00
MOVL C00125 BC00125 V=200.0 PL=0
REFP 3 C00126 BC00126
CALL JOB:SEARCH-R1
SET P0307 P0006
SFTON P0307
MOVL C00127 BC00127 V=166.7 PL=0
REFP 3 C00128 BC00128
CALL JOB:SEARCH-R1
SET P0307 P0006
SFTON P0307
MOVL C00129 BC00129 V=166.7 PL=0
SFTOF
'------------------------
'W15A L
'------------------------
SFTOF
MOVJ C00130 BC00130 VJ=50.00
MOVL C00131 BC00131 V=200.0 PL=0
REFP 3 C00132 BC00132
CALL JOB:SEARCH-R1
SET P0308 P0006
SFTON P0308
MOVL C00133 BC00133 V=166.7 PL=0
REFP 3 C00134 BC00134
CALL JOB:SEARCH-R1
SET P0308 P0006
SFTON P0308
MOVL C00135 BC00135 V=166.7 PL=0
SFTOF
'------------------------
'W15A P
'------------------------
SFTOF
MOVJ C00136 BC00136 VJ=50.00
MOVL C00137 BC00137 V=166.7 PL=0
REFP 3 C00138 BC00138
CALL JOB:SEARCH-R1
SET P0309 P0006
SFTON P0309
MOVL C00139 BC00139 V=166.7 PL=0
REFP 3 C00140 BC00140
CALL JOB:SEARCH-R1
SET P0309 P0006
SFTON P0309
MOVL C00141 BC00141 V=166.7 PL=0
SFTOF
MOVL C00142 BC00142 V=333.3
'------------------------
'W17A L
'------------------------
MOVL C00143 BC00143 V=500.0
SFTOF
MOVJ C00144 BC00144 VJ=20.00
MOVL C00145 BC00145 V=166.7 PL=0
REFP 3 C00146 BC00146
CALL JOB:SEARCH-R1
SET P0310 P0006
SFTON P0310
MOVL C00147 BC00147 V=166.7 PL=0
REFP 3 C00148 BC00148
CALL JOB:SEARCH-R1
SET P0310 P0006
SFTON P0310
MOVL C00149 BC00149 V=166.7 PL=0
SFTOF
'------------------------
'W17A P
'------------------------
SFTOF
MOVL C00150 BC00150 V=416.7
MOVL C00151 BC00151 V=166.7 PL=0
REFP 3 C00152 BC00152
CALL JOB:SEARCH-R1
SET P0311 P0006
SFTON P0311
MOVL C00153 BC00153 V=166.7 PL=0
REFP 3 C00154 BC00154
CALL JOB:SEARCH-R1
SET P0311 P0006
SFTON P0311
MOVL C00155 BC00155 V=166.7 PL=0
SFTOF
MOVJ C00156 BC00156 VJ=10.00
MOVJ C00157 BC00157 VJ=20.00
MOVJ C00158 BC00158 VJ=50.00
MOVJ C00159 BC00159 VJ=50.00
MOVJ C00160 BC00160 VJ=70.00
MOVJ C00161 BC00161 VJ=30.00
MOVJ C00162 BC00162 VJ=30.00
'------------------------
'------------------------
'LEWA STRONA PROFIL GORA
'------------------------
'------------------------
MOVJ C00163 BC00163 VJ=30.00
MOVJ C00164 BC00164 VJ=30.00
MOVJ C00165 BC00165 VJ=30.00
'------------------------
'W17B L
'------------------------
SFTOF
MOVJ C00166 BC00166 VJ=15.00
MOVL C00167 BC00167 V=166.7 PL=0
REFP 3 C00168 BC00168
CALL JOB:SEARCH-R1
SET P0350 P0006
SFTON P0350
MOVL C00169 BC00169 V=166.7 PL=0
REFP 3 C00170 BC00170
CALL JOB:SEARCH-R1
SET P0350 P0006
SFTON P0350
MOVL C00171 BC00171 V=166.7 PL=0
SFTOF
'------------------------
'W17B P
'------------------------
SFTOF
MOVL C00172 BC00172 V=333.3
MOVL C00173 BC00173 V=166.7 PL=0
REFP 3 C00174 BC00174
CALL JOB:SEARCH-R1
SET P0351 P0006
SFTON P0351
MOVL C00175 BC00175 V=166.7 PL=0
REFP 3 C00176 BC00176
CALL JOB:SEARCH-R1
SET P0351 P0006
SFTON P0351
MOVL C00177 BC00177 V=166.7 PL=0
SFTOF
'POPRAWID DOJAZD
'------------------------
'W15B L
'------------------------
SFTOF
MOVJ C00178 BC00178 VJ=10.00
MOVL C00179 BC00179 V=166.7 PL=0
REFP 3 C00180 BC00180
CALL JOB:SEARCH-R1
SET P0352 P0006
SFTON P0352
MOVL C00181 BC00181 V=166.7 PL=0
REFP 3 C00182 BC00182
CALL JOB:SEARCH-R1
SET P0352 P0006
SFTON P0352
MOVL C00183 BC00183 V=166.7 PL=0
SFTOF
'------------------------
'W15B P
'------------------------
SFTOF
MOVJ C00184 BC00184 VJ=20.00
MOVL C00185 BC00185 V=166.7 PL=0
REFP 3 C00186 BC00186
CALL JOB:SEARCH-R1
SET P0353 P0006
SFTON P0353
MOVL C00187 BC00187 V=166.7 PL=0
REFP 3 C00188 BC00188
CALL JOB:SEARCH-R1
SET P0353 P0006
SFTON P0353
MOVL C00189 BC00189 V=166.7 PL=0
SFTOF
'------------------------
'W18B L
'------------------------
SFTOF
MOVJ C00190 BC00190 VJ=50.00
MOVL C00191 BC00191 V=166.7 PL=0
REFP 3 C00192 BC00192
CALL JOB:SEARCH-R1
SET P0354 P0006
SFTON P0354
MOVL C00193 BC00193 V=166.7 PL=0
REFP 3 C00194 BC00194
CALL JOB:SEARCH-R1
SET P0354 P0006
SFTON P0354
MOVL C00195 BC00195 V=166.7 PL=0
SFTOF
'------------------------
'W18B P
'------------------------
SFTOF
MOVJ C00196 BC00196 VJ=50.00
MOVL C00197 BC00197 V=166.7 PL=0
REFP 3 C00198 BC00198
CALL JOB:SEARCH-R1
SET P0355 P0006
SFTON P0355
MOVL C00199 BC00199 V=166.7 PL=0
REFP 3 C00200 BC00200
CALL JOB:SEARCH-R1
SET P0355 P0006
SFTON P0355
MOVL C00201 BC00201 V=166.7 PL=0
SFTOF
'------------------------
'W13B L
'------------------------
SFTOF
MOVJ C00202 BC00202 VJ=50.00
MOVL C00203 BC00203 V=166.7 PL=0
REFP 3 C00204 BC00204
CALL JOB:SEARCH-R1
SET P0356 P0006
SFTON P0356
MOVL C00205 BC00205 V=166.7 PL=0
REFP 3 C00206 BC00206
CALL JOB:SEARCH-R1
SET P0356 P0006
SFTON P0356
MOVL C00207 BC00207 V=166.7 PL=0
SFTOF
'------------------------
'W13B P
'------------------------
SFTOF
MOVJ C00208 BC00208 VJ=50.00
MOVL C00209 BC00209 V=166.7 PL=0
REFP 3 C00210 BC00210
CALL JOB:SEARCH-R1
SET P0357 P0006
SFTON P0357
MOVL C00211 BC00211 V=166.7 PL=0
REFP 3 C00212 BC00212
CALL JOB:SEARCH-R1
SET P0357 P0006
SFTON P0357
MOVL C00213 BC00213 V=166.7 PL=0
SFTOF
'------------------------
'W19B L
'------------------------
SFTOF
MOVJ C00214 BC00214 VJ=50.00
MOVL C00215 BC00215 V=166.7 PL=0
REFP 3 C00216 BC00216
CALL JOB:SEARCH-R1
SET P0358 P0006
SFTON P0358
MOVL C00217 BC00217 V=166.7 PL=0
REFP 3 C00218 BC00218
CALL JOB:SEARCH-R1
SET P0358 P0006
SFTON P0358
MOVL C00219 BC00219 V=166.7 PL=0
SFTOF
'------------------------
'W19B P
'------------------------
SFTOF
MOVJ C00220 BC00220 VJ=50.00
MOVL C00221 BC00221 V=166.7 PL=0
REFP 3 C00222 BC00222
CALL JOB:SEARCH-R1
SET P0359 P0006
SFTON P0359
MOVL C00223 BC00223 V=166.7 PL=0
REFP 3 C00224 BC00224
CALL JOB:SEARCH-R1
SET P0359 P0006
SFTON P0359
MOVL C00225 BC00225 V=166.7 PL=0
SFTOF
'------------------------
'W14B L
'------------------------
SFTOF
MOVJ C00226 BC00226 VJ=50.00
MOVL C00227 BC00227 V=166.7 PL=0
REFP 3 C00228 BC00228
CALL JOB:SEARCH-R1
SET P0360 P0006
SFTON P0360
MOVL C00229 BC00229 V=166.7 PL=0
REFP 3 C00230 BC00230
CALL JOB:SEARCH-R1
SET P0360 P0006
SFTON P0360
MOVL C00231 BC00231 V=166.7 PL=0
SFTOF
'------------------------
'W14B P
'------------------------
SFTOF
MOVJ C00232 BC00232 VJ=50.00
MOVL C00233 BC00233 V=166.7 PL=0
REFP 3 C00234 BC00234
CALL JOB:SEARCH-R1
SET P0361 P0006
SFTON P0361
MOVL C00235 BC00235 V=166.7 PL=0
REFP 3 C00236 BC00236
CALL JOB:SEARCH-R1
SET P0361 P0006
SFTON P0361
MOVL C00237 BC00237 V=166.7 PL=0
SFTOF
MOVJ C00238 BC00238 VJ=50.00
MOVJ C00239 BC00239 VJ=50.00
MOVJ C00240 BC00240 VJ=50.00
MOVJ C00241 BC00241 VJ=50.00
MOVJ C00242 BC00242 VJ=50.00
'WELD
'WELD
'WELD
MOVJ C00243 BC00243 VJ=10.00
'**********************
'**********************
'POCZATEK SPAWANIA DOL
'**********************
'**********************
''
'**********************
'W1
'**********************
MOVJ C00244 BC00244 VJ=50.00
MOVJ C00245 BC00245 VJ=40.00
MOVL C00246 BC00246 V=166.7
SFTON P0104
MOVL C00247 BC00247 V=166.7
MACRO1 MJ#(0) ARGF24
ARCON
SFTON P0105
MOVL C00248 BC00248 V=11.7
ARCOF
SFTOF
MOVJ C00249 BC00249 VJ=20.00
MOVJ C00250 BC00250 VJ=30.00
MOVJ C00251 BC00251 VJ=50.00
MOVJ C00252 BC00252 VJ=40.00
MOVJ C00253 BC00253 VJ=20.00
'**********************
'W2
'**********************
SFTON P0108
MOVL C00254 BC00254 V=166.7
ARCON
SFTON P0109
MOVL C00255 BC00255 V=11.7
MOVL C00256 BC00256 V=11.7
ARCOF
SFTOF
MOVL C00257 BC00257 V=333.3
MOVJ C00258 BC00258 VJ=40.00
MOVJ C00259 BC00259 VJ=70.00
MOVJ C00260 BC00260 VJ=20.00
MOVL C00261 BC00261 V=666.7
'**********************
'W3
'**********************
SFTON P0101
MOVL C00262 BC00262 V=166.7
ARCON
SFTON P0100
MOVL C00263 BC00263 V=11.7
ARCOF
MOVL C00264 BC00264 V=166.7
SFTOF
MOVJ C00265 BC00265 VJ=30.00
MOVJ C00266 BC00266 VJ=30.00
MOVJ C00267 BC00267 VJ=50.00
MOVJ C00268 BC00268 VJ=30.00
MOVJ C00269 BC00269 VJ=40.00
'..................
'..................
'..................
'..................
' PROG SPAWANIE RAMA PRZED
MOVJ C00270 BC00270 VJ=50.00
MOVJ C00271 BC00271 VJ=25.00
CALL JOB:TWIN_5340_0ST_RAMA_PRZ_OBR1_SPAW
PAUSE
MOVJ C00272 BC00272 VJ=30.00
MOVJ C00273 BC00273 VJ=50.00
MOVJ C00274 BC00274 VJ=50.00
MOVJ C00275 BC00275 VJ=40.00
MOVJ C00276 BC00276 VJ=10.00
'**********************
'W9
'**********************
SFTON P0103
MACRO1 MJ#(0) ARGF24
MOVL C00277 BC00277 V=166.7
ARCON
SFTON P0102
MOVL C00278 BC00278 V=11.7
ARCOF
SFTOF
MOVL C00279 BC00279 V=166.7
MOVJ C00280 BC00280 VJ=40.00
MOVJ C00281 BC00281 VJ=70.00
MOVJ C00282 BC00282 VJ=50.00
MOVJ C00283 BC00283 VJ=20.00
'**********************
'W10
'**********************
MOVL C00284 BC00284 V=333.3
SFTON P0106
MOVL C00285 BC00285 V=166.7
ARCON
SFTON P0107
MOVL C00286 BC00286 V=11.7
ARCOF
SFTOF
MOVL C00287 BC00287 V=333.3
MOVJ C00288 BC00288 VJ=50.00
'**********************
'**********************
'POCZATEK SPAWANIA BOKI
'**********************
'**********************
MOVJ C00289 BC00289 VJ=50.00
MOVJ C00290 BC00290 VJ=50.00
'**********************
'W13A
'**********************
SFTON P0305
MOVL C00291 BC00291 V=250.0 PL=0
SFTOF
MACRO1 MJ#(0) ARGF10
ARCON
SFTON P0304
MOVL C00292 BC00292 V=10.8
ARCOF
SFTOF
MOVL C00293 BC00293 V=250.0
'W13B
MOVJ C00294 BC00294 VJ=30.00
MOVJ C00295 BC00295 VJ=50.00
MOVL C00296 BC00296 V=500.0
'**********************
'W13B
'**********************
SFTON P0356
MOVL C00297 BC00297 V=133.3 PL=0
SFTOF
ARCON
SFTON P0357
MOVL C00298 BC00298 V=10.8
ARCOF
SFTOF
MOVL C00299 BC00299 V=250.0
MOVJ C00300 BC00300 VJ=30.00
MOVJ C00301 BC00301 VJ=40.00
MOVJ C00302 BC00302 VJ=30.00
MOVJ C00303 BC00303 VJ=30.00
'**********************
'W14A
'**********************
MOVL C00304 BC00304 V=250.0
SFTON P0301
MOVL C00305 BC00305 V=50.0 PL=0
SFTOF
ARCON
SFTON P0300
MOVL C00306 BC00306 V=10.8
MOVL C00307 BC00307 V=10.8
MOVL C00308 BC00308 V=10.8
ARCOF
SFTOF
MOVL C00309 BC00309 V=150.0
MOVJ C00310 BC00310 VJ=40.00
MOVJ C00311 BC00311 VJ=30.00
MOVJ C00312 BC00312 VJ=30.00
MOVJ C00313 BC00313 VJ=30.00
MOVJ C00314 BC00314 VJ=30.00
'**********************
'W14B
'**********************
SFTON P0360
MOVL C00315 BC00315 V=333.3
MOVL C00316 BC00316 V=166.7 PL=0
SFTOF
ARCON
SFTON P0361
MOVL C00317 BC00317 V=10.8
MOVL C00318 BC00318 V=10.8
MOVL C00319 BC00319 V=10.8
ARCOF
SFTOF
MOVL C00320 BC00320 V=250.0
MOVJ C00321 BC00321 VJ=40.00
MOVJ C00322 BC00322 VJ=40.00
MOVJ C00323 BC00323 VJ=30.00
MOVJ C00324 BC00324 VJ=40.00
MOVJ C00325 BC00325 VJ=30.00
MOVJ C00326 BC00326 VJ=30.00
MOVJ C00327 BC00327 VJ=30.00
MOVJ C00328 BC00328 VJ=30.00
MOVJ C00329 BC00329 VJ=30.00
'**********************
'W15A
'**********************
SFTON P0309
MOVL C00330 BC00330 V=166.7
MOVL C00331 BC00331 V=166.7 PL=0
SFTOF
ARCON
SFTON P0308
MOVL C00332 BC00332 V=10.8
ARCOF
SFTOF
MOVL C00333 BC00333 V=150.0
MOVJ C00334 BC00334 VJ=30.00
MOVJ C00335 BC00335 VJ=50.00
MOVJ C00336 BC00336 VJ=50.00
MOVJ C00337 BC00337 VJ=50.00
MOVJ C00338 BC00338 VJ=50.00
MOVJ C00339 BC00339 VJ=50.00
'**********************
'W15B
'**********************
SFTON P0352
MOVL C00340 BC00340 V=250.0
MOVL C00341 BC00341 V=83.3 PL=0
SFTOF
ARCON
SFTON P0353
MOVL C00342 BC00342 V=10.8
ARCOF
MOVL C00343 BC00343 V=66.7
SFTOF
MOVJ C00344 BC00344 VJ=40.00
MOVJ C00345 BC00345 VJ=50.00
MOVJ C00346 BC00346 VJ=50.00
'BRAK W TEJ DLUGOSCI
'**********************
'W16A
'**********************
'**********************
'W16B
'**********************
'BRAK W TEJ DLUGOSCI
'**********************
'W17A
'**********************
MOVJ C00347 BC00347 VJ=50.00
MOVJ C00348 BC00348 VJ=50.00
'**********************
'W17A
'**********************
SFTON P0310
MOVL C00349 BC00349 V=333.3
MOVL C00350 BC00350 V=166.7 PL=0
SFTOF
ARCON
SFTON P0311
MOVL C00351 BC00351 V=10.8
ARCOF
SFTOF
MOVL C00352 BC00352 V=333.3
MOVJ C00353 BC00353 VJ=30.00
MOVJ C00354 BC00354 VJ=30.00
MOVJ C00355 BC00355 VJ=50.00
MOVJ C00356 BC00356 VJ=50.00
MOVJ C00357 BC00357 VJ=50.00
MOVJ C00358 BC00358 VJ=50.00
MOVJ C00359 BC00359 VJ=50.00
MOVJ C00360 BC00360 VJ=30.00
MOVJ C00361 BC00361 VJ=30.00
'**********************
'W17B
'**********************
SFTON P0351
MOVL C00362 BC00362 V=166.7
MOVL C00363 BC00363 V=166.7 PL=0
SFTOF
ARCON
SFTON P0350
MOVL C00364 BC00364 V=10.8
ARCOF
SFTOF
MOVL C00365 BC00365 V=250.0
MOVJ C00366 BC00366 VJ=30.00
MOVJ C00367 BC00367 VJ=30.00
MOVJ C00368 BC00368 VJ=30.00
MOVJ C00369 BC00369 VJ=30.00
MOVJ C00370 BC00370 VJ=40.00
'**********************
'W18A
'**********************
SFTON P0306
MOVL C00371 BC00371 V=333.3
MOVL C00372 BC00372 V=166.7 PL=0
SFTOF
ARCON
SFTON P0307
MOVL C00373 BC00373 V=10.8
ARCOF
SFTOF
MOVL C00374 BC00374 V=250.0
MOVJ C00375 BC00375 VJ=30.00
MOVJ C00376 BC00376 VJ=30.00
MOVJ C00377 BC00377 VJ=50.00
MOVJ C00378 BC00378 VJ=50.00
MOVJ C00379 BC00379 VJ=50.00
'**********************
'W18B
'**********************
SFTON P0355
MOVL C00380 BC00380 V=166.7
MOVL C00381 BC00381 V=166.7 PL=0
SFTOF
ARCON
SFTON P0354
MOVL C00382 BC00382 V=10.8
ARCOF
MOVL C00383 BC00383 V=250.0
SFTOF
MOVJ C00384 BC00384 VJ=30.00
MOVJ C00385 BC00385 VJ=30.00
MOVJ C00386 BC00386 VJ=40.00
MOVJ C00387 BC00387 VJ=50.00
MOVJ C00388 BC00388 VJ=30.00
'**********************
'W19A
'**********************
MOVL C00389 BC00389 V=166.7
SFTON P0303
MOVL C00390 BC00390 V=166.7 PL=0
SFTOF
ARCON
SFTON P0302
MOVL C00391 BC00391 V=10.8
ARCOF
SFTOF
MOVL C00392 BC00392 V=150.0
MOVJ C00393 BC00393 VJ=30.00
MOVJ C00394 BC00394 VJ=50.00
MOVJ C00395 BC00395 VJ=50.00
'**********************
'W19B
'**********************
SFTON P0358
MOVL C00396 BC00396 V=500.0
MOVL C00397 BC00397 V=166.7 PL=0
SFTOF
ARCON
SFTON P0359
MOVL C00398 BC00398 V=10.8
ARCOF
SFTOF
MOVL C00399 BC00399 V=250.0
MOVJ C00400 BC00400 VJ=40.00
MOVJ C00401 BC00401 VJ=50.00
CALL JOB:MOVE_OUT_OF_TUNNEL
END
